// SIMATIC S7-200 project (STEP 7-Micro/WIN), CPU 221 REL 01.10

SYMBOL_TABLE USER1
Start            I0.0
Stopp            I0.1
dc1              Q0.0
dc2              Q0.1
dc3              Q0.2
Den1             Q0.3
den2             Q0.4
den3             Q0.5
END_SYMBOL_TABLE

ORGANIZATION_BLOCK MAIN:OB1
TITLE=
BEGIN
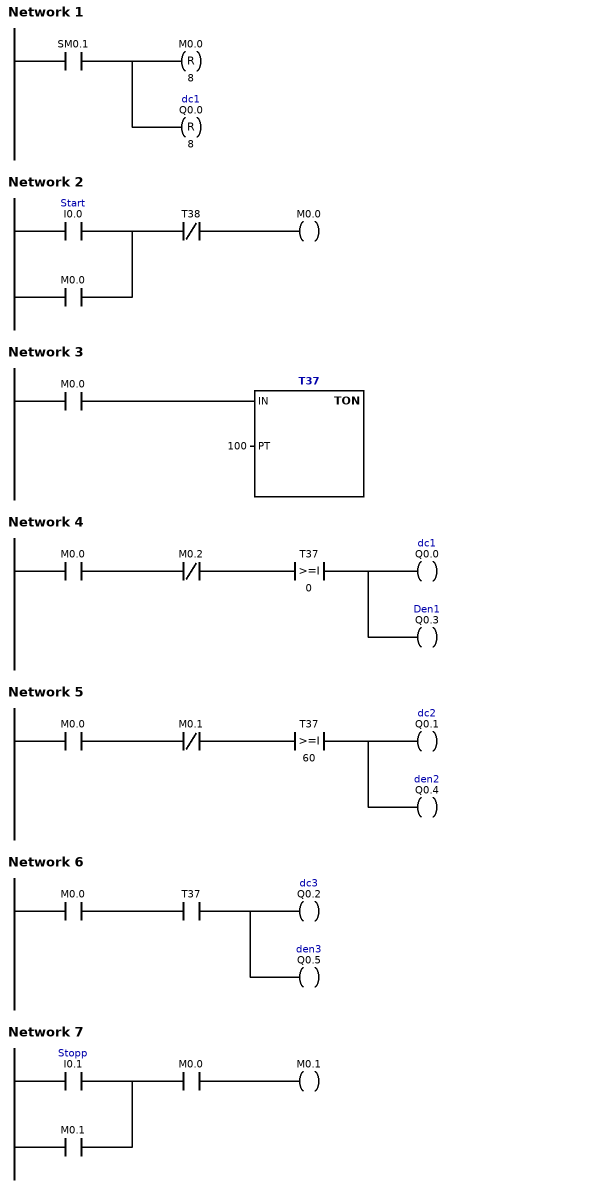
Network 1
LD     SM0.1
R      M0.0, 8
R      dc1:Q0.0, 8
Network 2
LD     Start:I0.0
O      M0.0
AN     T38
=      M0.0
Network 3
LD     M0.0
TON    T37, 100
Network 4
LD     M0.0
AN     M0.2
AW>=   T37, 0
=      dc1:Q0.0
=      Den1:Q0.3
Network 5
LD     M0.0
AN     M0.1
AW>=   T37, 60
=      dc2:Q0.1
=      den2:Q0.4
Network 6
LD     M0.0
A      T37
=      dc3:Q0.2
=      den3:Q0.5
Network 7
LD     Stopp:I0.1
O      M0.1
A      M0.0
=      M0.1
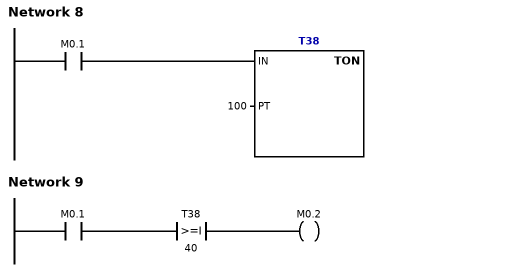
Network 8
LD     M0.1
TON    T38, 100
Network 9
LD     M0.1
AW>=   T38, 40
=      M0.2
END_ORGANIZATION_BLOCK
